// TIA Portal V17 export
// export: Created 2025-06-26T06:49:18.4879928Z, ExportSetting WithDefaults, DisplayName Totally Integrated Automation Portal, DisplayVersion V17 Update 8, DisplayName TIA Portal Openness, DisplayVersion V17 Update 8, DisplayName TIA Portal Version Control Interface, DisplayVersion V17, DisplayName STEP 7 Professional, DisplayVersion V17 Update 8, DisplayName STEP 7 Safety, DisplayVersion V17 Update 6, DisplayName WinCC Advanced, DisplayVersion V17 Update 8
FUNCTION "State1_Offline" : Void   // FC4, FBD
{ S7_Optimized_Access := 'TRUE' }
VERSION : 0.1
// stored: AutoNumber true, IsIECCheckEnabled false, SetENOAutomatically false, UDAEnableTagReadback false
   VAR_INPUT
      Active : Bool;
   END_VAR
   VAR_OUTPUT
      NextState : Bool;
   END_VAR
BEGIN

REGION Network 1: State number
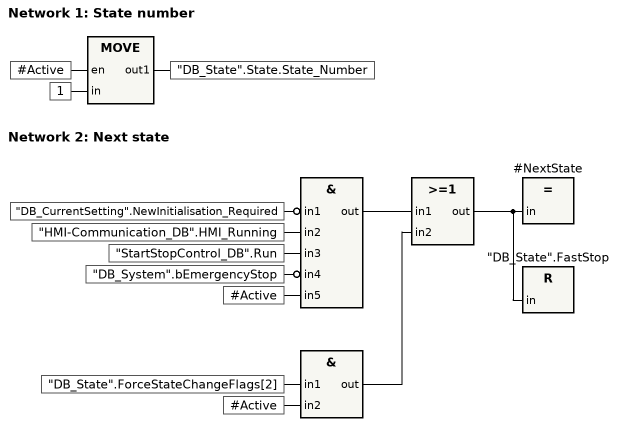
   IF #Active THEN "DB_State".State.State_Number := 1; END_IF;
END_REGION

REGION Network 2: Next state
   #NextState := (NOT "DB_CurrentSetting".NewInitialisation_Required AND "HMI-Communication_DB".HMI_Running AND "StartStopControl_DB".Run AND NOT "DB_System".bEmergencyStop AND #Active) OR ("DB_State".ForceStateChangeFlags[2] AND #Active);
   IF #NextState THEN "DB_State".FastStop := FALSE; END_IF;
END_REGION
END_FUNCTION
